// TIA Portal V17 export
// export: Created 2023-04-11T09:33:34.6239066Z, ExportSetting WithDefaults, DisplayName Totally Integrated Automation Portal, DisplayVersion V17 Update 3, DisplayName TIA Portal Openness, DisplayVersion V17 Update 3, DisplayName TIA Portal Version Control Interface, DisplayVersion V17, DisplayName SINAMICS Startdrive Advanced, DisplayVersion V17 Update2, DisplayName SINAMICS Startdrive G130, G150, S120, S150, SINAMICS MV, S210, DisplayVersion V17 Update2, DisplayName SINAMICS Startdrive G110M, G120, G120C, G120D, G120P, G115D, DisplayVersion V17 Update2, DisplayName STEP 7 Professional, DisplayVersion V17 Update 3, DisplayName STEP 7 Safety, DisplayVersion V17, DisplayName WinCC UA Professional, DisplayVersion V17 Update 3
FUNCTION "FC_aiPosSensor" : Void   // FC26, LAD
{ S7_Optimized_Access := 'TRUE' }
VERSION : 0.1
// stored: AutoNumber true, IsIECCheckEnabled false, SetENOAutomatically false, UDAEnableTagReadback false
   VAR_INPUT
      analogInt : Int;
      stroke : Real;
      limits : "t_aiPosSensorLimits";
   END_VAR
   VAR_IN_OUT
      sensorHandle : "t_aiPosSensor";
   END_VAR
BEGIN

REGION Network 1 (SCL)
   #sensorHandle.act := INT_TO_REAL(#analogInt) / 27648.0 * #stroke;
END_REGION

REGION Network 2
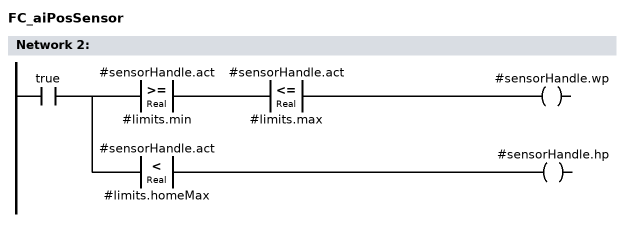
   RUNG wire#powerrail
      Contact( true )
      wire#w1
      { S7_Templates := "SrcType := Real" } GE_Contact(in1 := #sensorHandle.act, in2 := #limits.min)
      { S7_Templates := "SrcType := Real" } LE_Contact(in1 := #sensorHandle.act, in2 := #limits.max)
      Coil( #sensorHandle.wp )
   END_RUNG
   RUNG wire#w1
      { S7_Templates := "SrcType := Real" } LT_Contact(in1 := #sensorHandle.act, in2 := #limits.homeMax)
      Coil( #sensorHandle.hp )
   END_RUNG
   // the same network as SCL:
   #sensorHandle.wp := true AND (#sensorHandle.act >= #limits.min) AND (#sensorHandle.act <= #limits.max);
   #sensorHandle.hp := true AND (#sensorHandle.act < #limits.homeMax);
END_REGION
END_FUNCTION
